DATA_BLOCK "dbArchiveControlDoor"
{ S7_Optimized_Access := 'TRUE' }
VERSION : 0.8
NON_RETAIN
"fbArchiveControlDoor"

BEGIN

END_DATA_BLOCK

